FUNCTION_BLOCK ASRT_SR_AE_TO_SRT (* Composite FB for convert ASR + AE to ASRT *)
  (* Standard: 61499-2; Description: Copyright (c) 2026 HR Agrartechnik GmbH This program and the accompanying materials are made available under the terms of the Eclipse Public License 2.0 which is available at https://www.eclipse.org/legal/epl-2.0/ SPDX-License-Identifier: EPL-2.0 *)
  (* Version 1.0, 2026-09-06, Franz Höpfinger, HR Agrartechnik GmbH *)
  PACKAGE adapter::conversion::unidirectional;
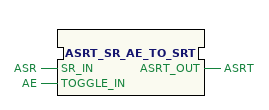
  SOCKETS
    SR_IN : adapter::types::unidirectional::ASR; (* Set/Reset Input *)
    TOGGLE_IN : adapter::types::unidirectional::AE; (* Toggle / Switch output *)
  END_SOCKETS
  PLUGS
    ASRT_OUT : adapter::types::unidirectional::ASRT; (* Adapter Output *)
  END_PLUGS
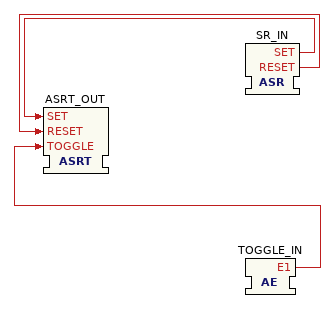
  EVENT_CONNECTIONS
    SR_IN.SET TO ASRT_OUT.SET;
    SR_IN.RESET TO ASRT_OUT.RESET;
    TOGGLE_IN.E1 TO ASRT_OUT.TOGGLE;
  END_CONNECTIONS
END_FUNCTION_BLOCK
